FUNCTION_BLOCK EL1094
VAR
	_io : EL1xx4_Data;
	{attribute addProperty Name "WcState"}
	_wcState : WcStateInputToggle;
	{attribute addProperty Name "Info data"}
	_infoData : InfoDataBase;
END_VAR

PROPERTY IO : REFERENCE TO EL1xx4_Data
GET
IO REF= _io;
END_GET
END_PROPERTY

PROPERTY WcState : REFERENCE TO WcStateInputToggle
GET
WcState REF= _wcState;
END_GET
END_PROPERTY

END_FUNCTION_BLOCK

(* stored: Version 1.1.0.1, ProductVersion 3.1.4024.9
   POU EL1094: Id {98213398-a337-0f50-004a-676f6db887d3}, SpecialFunc None
   Property IO: Id {186b9f06-5bdc-0b15-0599-65d43a145bdb}
   Get Get: Id {59b3c58e-35e8-00d9-0189-5f83e7c54fbe}
   Property WcState: Id {1061f7e7-520b-0825-0f92-f0937e23d521}
   Get Get: Id {4c99ced8-f843-0d1d-3c6d-4c4111aa1bc4} *)
